// LS Electric XG5000 project: 71회예상1_3
// PLC NewPLC
// module base 0 slot 0: 입출력 모듈:XBC-DR20S (DC 24V 입력 12점, 릴레이 출력 8점)

PROGRAM NewProgram (task: 스캔 프로그램)

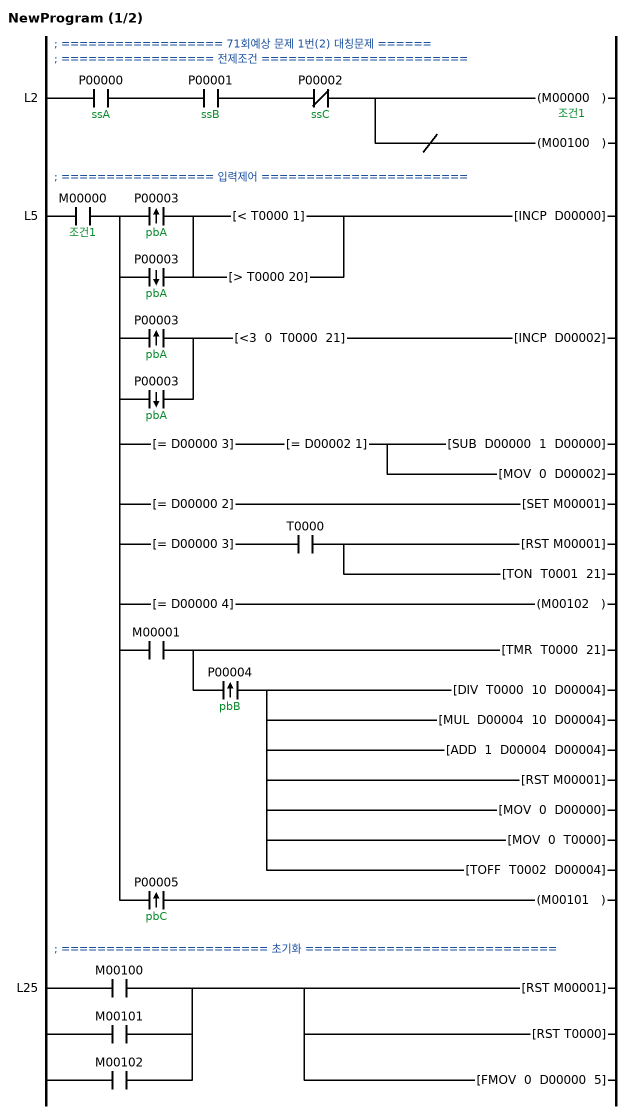
// ================== 71회예상 문제 1번(2) 대칭문제 ======
// ================= 전제조건 =======================
; L2
LOAD      P00000	// ssA
AND       P00001	// ssB
AND NOT   P00002	// ssC
OUT       M00000	// 조건1
NOT
OUT       M00100
// ================= 입력제어 =======================
; L5
LOAD      M00000	// 조건1
MPUSH
LOADP     P00003	// pbA
ORN       P00003	// pbA
AND LOAD
LOAD<     T0000 1
OR>       T0000 20
AND LOAD
INCP      D00000
MLOAD
LOADP     P00003	// pbA
ORN       P00003	// pbA
AND LOAD
AND<3     0 T0000 21
INCP      D00002
MLOAD
AND=      D00000 3
AND=      D00002 1
SUB       D00000 1 D00000
MOV       0 D00002
MLOAD
AND=      D00000 2
SET       M00001
MLOAD
AND=      D00000 3
AND       T0000
RST       M00001
TON       T0001 21
MLOAD
AND=      D00000 4
OUT       M00102
MLOAD
AND       M00001
TMR       T0000 21
ANDP      P00004	// pbB
DIV       T0000 10 D00004
MUL       D00004 10 D00004
ADD       1 D00004 D00004
RST       M00001
MOV       0 D00000
MOV       0 T0000
TOFF      T0002 D00004
MPOP
ANDP      P00005	// pbC
OUT       M00101
// ======================= 초기화 ============================
; L25
LOAD      M00100
OR        M00101
OR        M00102
RST       M00001
RST       T0000
FMOV      0 D00000 5

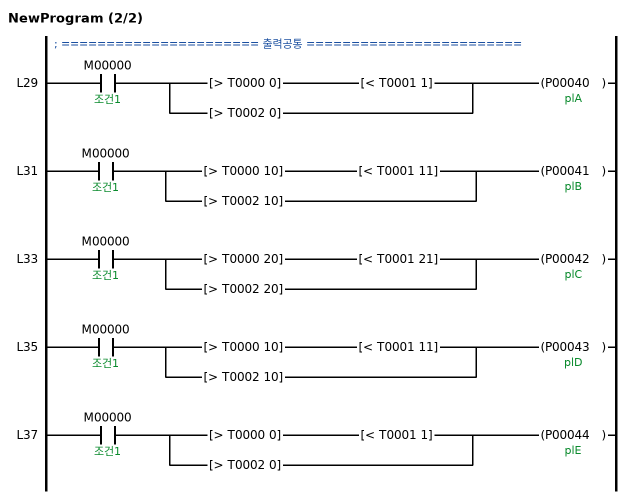
// ====================== 출력공통 ========================
; L29
LOAD      M00000	// 조건1
LOAD>     T0000 0
AND<      T0001 1
OR>       T0002 0
AND LOAD
OUT       P00040	// plA
; L31
LOAD      M00000	// 조건1
LOAD>     T0000 10
AND<      T0001 11
OR>       T0002 10
AND LOAD
OUT       P00041	// plB
; L33
LOAD      M00000	// 조건1
LOAD>     T0000 20
AND<      T0001 21
OR>       T0002 20
AND LOAD
OUT       P00042	// plC
; L35
LOAD      M00000	// 조건1
LOAD>     T0000 10
AND<      T0001 11
OR>       T0002 10
AND LOAD
OUT       P00043	// plD
; L37
LOAD      M00000	// 조건1
LOAD>     T0000 0
AND<      T0001 1
OR>       T0002 0
AND LOAD
OUT       P00044	// plE